VAR_GLOBAL CONSTANT
	nInitialize: SINT := 0;
	nStep: SINT := 1;
END_VAR

(* stored: Version 1.1.0.1, ProductVersion 3.1.4024.9
   GVL GVL_ZeroSpanCalibration: Id {bb8c3462-cd3c-4f34-a40a-a3bc9674890c} *)
